{attribute addProperty BoxType "EK1100-0000-0018"}
{attribute addProperty Id "Beckhoff_EL66xxEK1122Beckhoff_EL66xxEK1122_D63A030B1960245A_0001_EL6601_0000_0000EL6601_194A340D8010A_0002_EL6601_0000_0001EL6601_194A340D8010A_0003_EL6601_0000_0016EL6601_194A340D8010A_0004_EL6601_0000_0017EL6601_194A340D8010A_0005_EL6601_0000_0018EL6601_194A340D8010A_0006_EL6601_0000_0019EL6601_194A340D8010A_0007_EL6601_0000_0021EL6601_194A340D8010A_0008_EL6614_0000_0016EL6614_194A340D8010A_0009_EL6614_0000_0017EL6614_194A340D8010A_0010_EL6614_0000_0018EL6614_194A340D8010A_0011_EL6614_0000_0019EL6614_194A340D8010A_0012_EL6614_0000_0021EL6614_194A340D8010A_0013_EL6631_0000_0016EL6631_8C99EE5012816A_0014_EL6631_0000_0017EL6631_8C99EE5012816A_0015_EL6631_0000_0018EL6631_8C99EE5012816A_0016_EL6631_0010_0016EL6631_8C99EE5012816A_0017_EL6631_0010_0017EL6631_8C99EE5012816A_0018_EL6631_0010_0018EL6631_8C99EE5012816A_0019_EL6652_0000_0017EL6652_8C99EE5012816A_0020_EL6652_0000_0018EL6652_8C99EE5012816A_0021_EL6652_0010_0017EL6652_8C99EE5012816A_0022_EL6652_0010_0018EL6652_8C99EE5012816A_0023_EL6688_0000_0016EL6688_D8DFB0C717822.25A_0024_EL6688_0000_0017EL6688_CA73E61333842.25A_0025_EL6688_0000_0018EL6688_CA73E61333842.25A_0026_EL6688_0000_0019EL6688_CA73E61333842.25A_0027_EL6688_0000_0020EL6688_CA73E61333842.25A_0028_EL6688_0000_0022EL6688_092E4D1F33842.25A_0029_EL6690_0001_0000EL6690_0A78979B9011.25A_0030_EL6690_0001_0016EL6690_0A78979B9011.25A_0031_EL6690_0001_0017EL6690_0A78979B9011.25A_0037_EL6692_0000_0016EL6692_4FA89B0317822.25A_0038_EL6692_0000_0017EL6692_4FA89B0317822.25A_0039_EL6692_0000_0018EL6692_67810D9517822.25A_0045_EL6695_0000_0001EL6695_E3EE093115419.25A_0047_EL6695_0000_0002EL6695_E3EE093115419.25A_0049_EL6695_0000_0003EL6695_E3EE093115419.25A_0051_EL6695_0000_0004EL6695_5B9A4EC315419.25A_0053_EL6695_0000_0005EL6695_5B9A4EC315419.25A_0055_EL6695_0000_0006EL6695_5B9A4EC315419.25"}
{attribute addProperty CRC "3252810608"}
{attribute addProperty SizeInBites "7796"}
{attribute addProperty SizeInBytes "974.5"}
TYPE Beckhoff_EL66xx_C1E1F370 EXTENDS EK1100_179A0949 :
STRUCT
	{attribute addProperty Name "Beckhoff_EL66xxEK1122"}
	Beckhoff_EL66xxEK1122 : Beckhoff_EL66xxEK1122_D63A030B;
	{attribute addProperty Name "A_0001_EL6601_0000_0000"}
	A_0001_EL6601_0000_0000 : EL6601_194A340D;
	{attribute addProperty Name "A_0002_EL6601_0000_0001"}
	A_0002_EL6601_0000_0001 : EL6601_194A340D;
	{attribute addProperty Name "A_0003_EL6601_0000_0016"}
	A_0003_EL6601_0000_0016 : EL6601_194A340D;
	{attribute addProperty Name "A_0004_EL6601_0000_0017"}
	A_0004_EL6601_0000_0017 : EL6601_194A340D;
	{attribute addProperty Name "A_0005_EL6601_0000_0018"}
	A_0005_EL6601_0000_0018 : EL6601_194A340D;
	{attribute addProperty Name "A_0006_EL6601_0000_0019"}
	A_0006_EL6601_0000_0019 : EL6601_194A340D;
	{attribute addProperty Name "A_0007_EL6601_0000_0021"}
	A_0007_EL6601_0000_0021 : EL6601_194A340D;
	{attribute addProperty Name "A_0008_EL6614_0000_0016"}
	A_0008_EL6614_0000_0016 : EL6614_194A340D;
	{attribute addProperty Name "A_0009_EL6614_0000_0017"}
	A_0009_EL6614_0000_0017 : EL6614_194A340D;
	{attribute addProperty Name "A_0010_EL6614_0000_0018"}
	A_0010_EL6614_0000_0018 : EL6614_194A340D;
	{attribute addProperty Name "A_0011_EL6614_0000_0019"}
	A_0011_EL6614_0000_0019 : EL6614_194A340D;
	{attribute addProperty Name "A_0012_EL6614_0000_0021"}
	A_0012_EL6614_0000_0021 : EL6614_194A340D;
	{attribute addProperty Name "A_0013_EL6631_0000_0016"}
	A_0013_EL6631_0000_0016 : EL6631_8C99EE50;
	{attribute addProperty Name "A_0014_EL6631_0000_0017"}
	A_0014_EL6631_0000_0017 : EL6631_8C99EE50;
	{attribute addProperty Name "A_0015_EL6631_0000_0018"}
	A_0015_EL6631_0000_0018 : EL6631_8C99EE50;
	{attribute addProperty Name "A_0016_EL6631_0010_0016"}
	A_0016_EL6631_0010_0016 : EL6631_8C99EE50;
	{attribute addProperty Name "A_0017_EL6631_0010_0017"}
	A_0017_EL6631_0010_0017 : EL6631_8C99EE50;
	{attribute addProperty Name "A_0018_EL6631_0010_0018"}
	A_0018_EL6631_0010_0018 : EL6631_8C99EE50;
	{attribute addProperty Name "A_0019_EL6652_0000_0017"}
	A_0019_EL6652_0000_0017 : EL6652_8C99EE50;
	{attribute addProperty Name "A_0020_EL6652_0000_0018"}
	A_0020_EL6652_0000_0018 : EL6652_8C99EE50;
	{attribute addProperty Name "A_0021_EL6652_0010_0017"}
	A_0021_EL6652_0010_0017 : EL6652_8C99EE50;
	{attribute addProperty Name "A_0022_EL6652_0010_0018"}
	A_0022_EL6652_0010_0018 : EL6652_8C99EE50;
	{attribute addProperty Name "A_0023_EL6688_0000_0016"}
	A_0023_EL6688_0000_0016 : EL6688_D8DFB0C7;
	{attribute addProperty Name "A_0024_EL6688_0000_0017"}
	A_0024_EL6688_0000_0017 : EL6688_CA73E613;
	{attribute addProperty Name "A_0025_EL6688_0000_0018"}
	A_0025_EL6688_0000_0018 : EL6688_CA73E613;
	{attribute addProperty Name "A_0026_EL6688_0000_0019"}
	A_0026_EL6688_0000_0019 : EL6688_CA73E613;
	{attribute addProperty Name "A_0027_EL6688_0000_0020"}
	A_0027_EL6688_0000_0020 : EL6688_CA73E613;
	{attribute addProperty Name "A_0028_EL6688_0000_0022"}
	A_0028_EL6688_0000_0022 : EL6688_092E4D1F;
	{attribute addProperty Name "A_0029_EL6690_0001_0000"}
	A_0029_EL6690_0001_0000 : EL6690_0A78979B;
	{attribute addProperty Name "A_0030_EL6690_0001_0016"}
	A_0030_EL6690_0001_0016 : EL6690_0A78979B;
	{attribute addProperty Name "A_0031_EL6690_0001_0017"}
	A_0031_EL6690_0001_0017 : EL6690_0A78979B;
	{attribute addProperty Name "A_0037_EL6692_0000_0016"}
	A_0037_EL6692_0000_0016 : EL6692_4FA89B03;
	{attribute addProperty Name "A_0038_EL6692_0000_0017"}
	A_0038_EL6692_0000_0017 : EL6692_4FA89B03;
	{attribute addProperty Name "A_0039_EL6692_0000_0018"}
	A_0039_EL6692_0000_0018 : EL6692_67810D95;
	{attribute addProperty Name "A_0045_EL6695_0000_0001"}
	A_0045_EL6695_0000_0001 : EL6695_E3EE0931;
	{attribute addProperty Name "A_0047_EL6695_0000_0002"}
	A_0047_EL6695_0000_0002 : EL6695_E3EE0931;
	{attribute addProperty Name "A_0049_EL6695_0000_0003"}
	A_0049_EL6695_0000_0003 : EL6695_E3EE0931;
	{attribute addProperty Name "A_0051_EL6695_0000_0004"}
	A_0051_EL6695_0000_0004 : EL6695_5B9A4EC3;
	{attribute addProperty Name "A_0053_EL6695_0000_0005"}
	A_0053_EL6695_0000_0005 : EL6695_5B9A4EC3;
	{attribute addProperty Name "A_0055_EL6695_0000_0006"}
	A_0055_EL6695_0000_0006 : EL6695_5B9A4EC3;
END_STRUCT
END_TYPE

(* stored: Version 1.2.0.0, ProductVersion 3.1.4024.9
   DUT Beckhoff_EL66xx_C1E1F370: Id {7bddc5b7-5e74-40a3-b508-0dfb403b6f55} *)
